KUKA KRL program: letter_m_surname.src

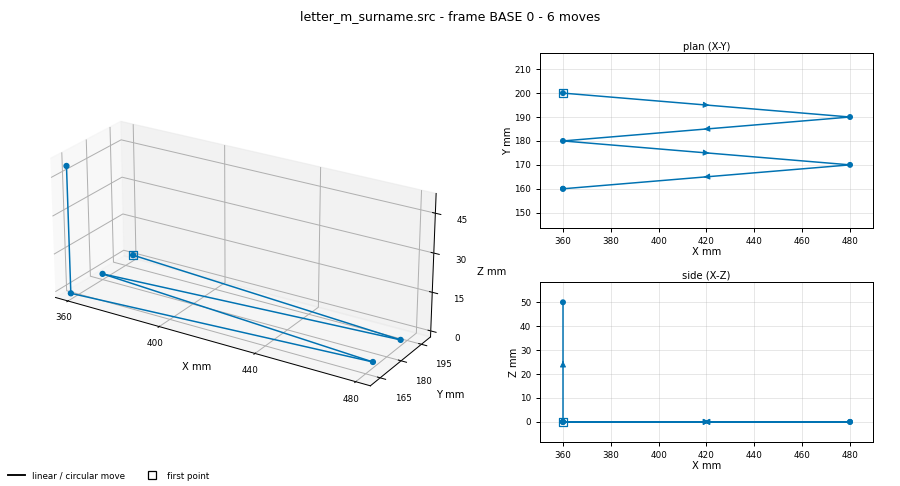
[picture p0: tool path of letter_m_surname.src in frame BASE 0, 6 of 9 moves have a stored position in this frame; points joined in program order, loops and branches not executed]
&ACCESS RVP
&REL 1
&PARAM TEMPLATE = C:\KRC\Roboter\Template\vorgabe
&PARAM EDITMASK = *
DEF letter_m_surname ( )

;FOLD Initialise and set default speed
BAS (#INITMOV,0)
BAS (#VEL_PTP,100)
BAS (#ACC_PTP,20)
$VEL.CP=0.2
BAS (#TOOL,0)
BAS (#BASE,0)
;ENDFOLD

$ADVANCE = 5

; Program generated by RoboDK v5.2.5 for KUKA KR 4 R600 on 07/01/2025 12:35:09
; Using nominal kinematics.
$VEL.CP = 0.10000
PTP {A1 0.00000,A2 -101.70200,A3 131.55600,A4 0.00000,A5 60.14530,A6 0.00000,E1 0.00000}
PTP {A1 -35.53770,A2 -48.63810,A3 112.93800,A4 0.00000,A5 25.70030,A6 -35.53770,E1 0.00000}
$VEL.CP = 0.05000
LIN {X 360.000,Y 200.000,Z 0.000,A 0.000,B 0.000,C 0.000,E1 0.00000}
$VEL.CP = 0.07500
LIN {X 480.000,Y 190.000,Z 0.000,A 0.000,B 0.000,C 0.000,E1 0.00000}
LIN {X 360.000,Y 180.000,Z 0.000,A 0.000,B 0.000,C 0.000,E1 0.00000}
LIN {X 480.000,Y 170.000,Z 0.000,A 0.000,B 0.000,C 0.000,E1 0.00000}
LIN {X 360.000,Y 160.000,Z 0.000,A 0.000,B 0.000,C 0.000,E1 0.00000}
$VEL.CP = 0.05000
LIN {X 360.000,Y 160.000,Z 50.000,A 0.000,B 0.000,C 0.000,E1 0.00000}
$VEL.CP = 0.10000
PTP {A1 0.00000,A2 -101.70200,A3 131.55600,A4 0.00000,A5 60.14530,A6 0.00000,E1 0.00000}
END
